// TIA Portal V17 export
// export: Created 2025-03-10T13:13:21.0797251Z, ExportSetting WithDefaults, DisplayName Totally Integrated Automation Portal, DisplayVersion V17 Update 8, DisplayName TIA Portal Openness, DisplayVersion V17 Update 8, DisplayName TIA Portal Version Control Interface, DisplayVersion V17, DisplayName SINAMICS Startdrive Advanced, DisplayVersion V17 SP2, DisplayName SINAMICS Startdrive G110M, G120, G120C, G120D, G120P, G115D, DisplayVersion V17 SP2, DisplayName SINAMICS Startdrive G130, G150, S120, S150, SINAMICS MV, S210, DisplayVersion V17 SP2, DisplayName STEP 7 Professional, DisplayVersion V17 Update 8, DisplayName SINUMERIK ONE STEP 7 Toolbox, DisplayVersion V17 Update 12, DisplayName SINUMERIK 840D sl STEP 7 Toolbox, DisplayVersion V17 Update 12, DisplayName STEP 7 Safety, DisplayVersion V17 Update 6, DisplayName WinCC Advanced, DisplayVersion V17 Update 8
TYPE "LOAD FEEDER SEQUENCE"
// stored: IsFailsafeCompliant false
   STRUCT
      "START GENERAL CONDITIONS" : Bool;   // General Conditions
      "START INITIAL CONDITIONS" : Bool;   // Initial Conditions
      "START SEMI REQUEST" : Bool;   // Semi Start Request
      "START AUTO REQUEST" : Bool;   // Auto Start Request
      "START COMMAND" : Bool;   // Global Start Request
      "STOP GENERAL CONDITIONS" : Bool;   // General Conditions
      "STOP INITIAL CONDITIONS" : Bool;   // Initial Conditions
      "STOP SEMI REQUEST" : Bool;   // Semi Start Request
      "STOP AUTO REQUEST" : Bool;   // Auto Start Request
      "STOP COMMAND" : Bool;   // Global Start Request
      "SEQUENCE RUNNING" : Bool;   // Sequence Running
      "STEP 1" : Bool;   // Step 1
      "STEP 2" : Bool;   // Step 2
      "STEP 3" : Bool;   // Step 3
      "STEP 4" : Bool;   // Step 4
      "STEP 5" : Bool;   // Step 5
      "STEP 6" : Bool;   // Step 6
      "STEP 7" : Bool;   // Step 7
      "RESET PLC SEQUENCE" : Bool;   // Reset PLC Sequence
      "REQUEST START VALVE" : Bool;   // Semi Auto Request
      "REQUEST STOP VALVE" : Bool;
      "REQUEST START PRESSURE" : Bool;   // Semi Auto Request
      "REQUESTE STOP PRESSURE" : Bool;
      "SETPOINT PRESSURE" : Real;
      "PASS STEP" : Bool;
      "SEQUENCE DONE" : Bool;   // Sequence Done
      WARNING : Bool;   // Warning
      "START GENERAL CONDITIONS HELP" : Bool;   // General Conditions Help
      "START INITIAL CONDITIONS HELP" : Bool;   // Initial Conditions Help
      "STOP GENERAL CONDITIONS HELP" : Bool;   // General Conditions Help
      "STOP INITIAL CONDITIONS HELP" : Bool;   // Initial Conditions Help
      "WARNING GONE" : Bool;   // Warning Gone
      "TIME ACTION" : Time;
      "APPLIED TIME ACTION" : Bool;
      "HMI START CONDITIONS" : Bool;   // HMI Start Conditions
      "HMI STOP CONDITIONS" : Bool;   // HMI Stop Conditions
      "HMI SEQUENCE RUNNING" : Bool;   // HMI Sequence Running
      "HMI SEQUENCE DONE" : Bool;   // HMI Sequence Done
      "HMI TIME LOAD" : UDInt;   // HMI Time Load
      "HMI FEEDBACK TIMER LOAD" : Int;
   END_STRUCT;
END_TYPE
